// TIA Portal V15.1 export
// export: Created 2020-06-12T07:35:43.4599609Z, ExportSetting None, DisplayName Totally Integrated Automation Portal, DisplayVersion V15.1, DisplayName TIA Portal Openness, DisplayVersion V15.1, DisplayName STEP 7 Professional, DisplayVersion V15.1, DisplayName STEP 7 Safety, DisplayVersion V15.1, DisplayName WinCC Advanced, DisplayVersion V15.1
FUNCTION "CW_Call" : Void   // FC142, FBD
TITLE = Cooling water call
{ S7_Optimized_Access := 'TRUE' }
// stored: SetENOAutomatically False
BEGIN

REGION Network 1: Cooling common signals
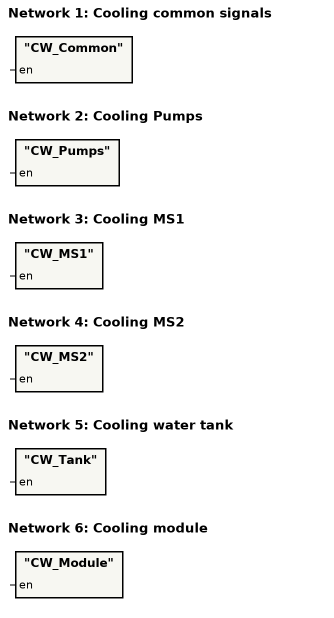
   "CW_Common"();
END_REGION

REGION Network 2: Cooling Pumps
   "CW_Pumps"();
END_REGION

REGION Network 3: Cooling MS1
   "CW_MS1"();
END_REGION

REGION Network 4: Cooling MS2
   "CW_MS2"();
END_REGION

REGION Network 5: Cooling water tank
   "CW_Tank"();
END_REGION

REGION Network 6: Cooling module
   "CW_Module"();
END_REGION
END_FUNCTION
